FUNCTION GetAngleDegreesFrom3Sides : LREAL
VAR_INPUT
	adjacentLeft : LREAL;
	opposite : LREAL;
	adjacentRight : LREAL;
END_VAR
VAR
	cosTargetAngle : LREAL;
	targetAngleRadians : LREAL;
END_VAR

//Cosine formula
cosTargetAngle := ((adjacentLeft * adjacentLeft) + (adjacentRight * adjacentRight) - (opposite * opposite))
				  /
				  (2 * adjacentLeft * adjacentRight);
				  
targetAngleRadians := ACOS(cosTargetAngle);

GetAngleDegreesFrom3Sides := RadiansToDegrees(targetAngleRadians);

END_FUNCTION

(* stored: Version 1.1.0.1, ProductVersion 3.1.4024.12
   POU GetAngleDegreesFrom3Sides: Id {481ddc49-b5a4-45fc-9931-09f4136c6205}, SpecialFunc None *)
